LIN {X 0,Y 58.147,Z 234.055,A -85,B 0,C 180,E1 -29041.086,E2 -29041.086} C_VEL
LIN {X 0,Y 58.532,Z 233.998,A -85,B 0,C 180,E1 -29053.833,E2 -29053.833} C_VEL
LIN {X 0,Y 58.812,Z 233.964,A -85,B 0,C 180,E1 -29063.136,E2 -29063.136} C_VEL
LIN {X 0,Y 59.332,Z 233.898,A -85,B 0,C 180,E1 -29069.999,E2 -29069.999} C_VEL
LIN {X 0,Y 59.001,Z 234.006,A -85,B 0,C 180,E1 -29073.2,E2 -29073.2} C_VEL
LIN {X 0,Y 60.875,Z 241.106,A -85,B 0,C 180,E1 -29076.628,E2 -29076.628} C_VEL
LIN {X 0,Y 61.421,Z 249.605,A -85,B 0,C 180,E1 -29080.715,E2 -29080.715} C_VEL
LIN {X 0,Y 61.771,Z 259.733,A -85,B 0,C 180,E1 -29086.524,E2 -29086.524} C_VEL
LIN {X 0,Y 59.443,Z 268.589,A -85,B 0,C 180,E1 -29092.592,E2 -29092.592} C_VEL
LIN {X 0,Y 57.484,Z 276.014,A -85,B 0,C 180,E1 -29099.276,E2 -29099.276} C_VEL
LIN {X 0,Y 56.132,Z 282.39,A -85,B 0,C 180,E1 -29106.678,E2 -29106.678} C_VEL
LIN {X 0,Y 55.622,Z 288.326,A -85,B 0,C 180,E1 -29115.356,E2 -29115.356} C_VEL
LIN {X 0,Y 56.401,Z 293.902,A -85,B 0,C 180,E1 -29125.519,E2 -29125.519} C_VEL
LIN {X 0,Y 58.844,Z 298.13,A -85,B 0,C 180,E1 -29135.112,E2 -29135.112} C_VEL
LIN {X 0,Y 62.731,Z 301.206,A -85,B 0,C 180,E1 -29143.717,E2 -29143.717} C_VEL
LIN {X 0,Y 65.186,Z 302.377,A -85,B 0,C 180,E1 -29147.553,E2 -29147.553} C_VEL
LIN {X 0,Y 69.185,Z 303.56,A -85,B 0,C 180,E1 -29152.557,E2 -29152.557} C_VEL
LIN {X 0,Y 71.068,Z 304.167,A -85,B 0,C 180,E1 -29155.394,E2 -29155.394} C_VEL
LIN {X 0,Y 73.084,Z 304.818,A -85,B 0,C 180,E1 -29160.5,E2 -29160.5} C_VEL
LIN {X 0,Y 75.674,Z 305.088,A -85,B 0,C 180,E1 -29165.303,E2 -29165.303} C_VEL
LIN {X 0,Y 78.302,Z 305.043,A -85,B 0,C 180,E1 -29167.536,E2 -29167.536} C_VEL
LIN {X 0,Y 86.056,Z 304.44,A -85,B 0,C 180,E1 -29171.478,E2 -29171.478} C_VEL
LIN {X 0,Y 87.267,Z 304.356,A -85,B 0,C 180,E1 -29173.985,E2 -29173.985} C_VEL
LIN {X 0,Y 87.254,Z 304.599,A -85,B 0,C 180,E1 -29178.799,E2 -29178.799} C_VEL
LIN {X 0,Y 86.938,Z 305.009,A -85,B 0,C 180,E1 -29183.845,E2 -29183.845} C_VEL
LIN {X 0,Y 86.523,Z 305.313,A -85,B 0,C 180,E1 -29186.685,E2 -29186.685} C_VEL
LIN {X 0,Y 85.779,Z 305.678,A -85,B 0,C 180,E1 -29189.449,E2 -29189.449} C_VEL
LIN {X 0,Y 82.562,Z 306.32,A -85,B 0,C 180,E1 -29191.655,E2 -29191.655} C_VEL
LIN {X 0,Y 76.874,Z 306.876,A -85,B 0,C 180,E1 -29194.635,E2 -29194.635} C_VEL
LIN {X 0,Y 66.462,Z 306.835,A -85,B 0,C 180,E1 -29202.252,E2 -29202.252} C_VEL
LIN {X 0,Y 61.77,Z 306.092,A -85,B 0,C 180,E1 -29206.949,E2 -29206.949} C_VEL
LIN {X 0,Y 57.805,Z 304.93,A -85,B 0,C 180,E1 -29212.563,E2 -29212.563} C_VEL
LIN {X 0,Y 53.214,Z 302.399,A -85,B 0,C 180,E1 -29222.469,E2 -29222.469} C_VEL
LIN {X 0,Y 50.575,Z 298.791,A -85,B 0,C 180,E1 -29233.865,E2 -29233.865} C_VEL
LIN {X 0,Y 50.036,Z 293.872,A -85,B 0,C 180,E1 -29245.974,E2 -29245.974} C_VEL
LIN {X 0,Y 49.816,Z 288.545,A -85,B 0,C 180,E1 -29255.483,E2 -29255.483} C_VEL
LIN {X 0,Y 50.428,Z 282.817,A -85,B 0,C 180,E1 -29263.704,E2 -29263.704} C_VEL
LIN {X 0,Y 51.962,Z 275.543,A -85,B 0,C 180,E1 -29271.837,E2 -29271.837} C_VEL
LIN {X 0,Y 52.516,Z 271.35,A -85,B 0,C 180,E1 -29275.783,E2 -29275.783} C_VEL
LIN {X 0,Y 53.107,Z 261.909,A -85,B 0,C 180,E1 -29282.979,E2 -29282.979} C_VEL
LIN {X 0,Y 53.75,Z 253.089,A -85,B 0,C 180,E1 -29288.314,E2 -29288.314} C_VEL
LIN {X 0,Y 54.341,Z 243.271,A -85,B 0,C 180,E1 -29292.972,E2 -29292.972} C_VEL
LIN {X 0,Y 54.24,Z 241.536,A -85,B 0,C 180,E1 -29293.788,E2 -29293.788} C_VEL
LIN {X 0,Y 51.257,Z 235.226,A -85,B 0,C 180,E1 -29297.691,E2 -29297.691} C_VEL
LIN {X 0,Y 51.188,Z 234.914,A -85,B 0,C 180,E1 -29297.945,E2 -29297.945} C_VEL
LIN {X 0,Y 51.071,Z 234.929,A -85,B 0,C 180,E1 -29306.594,E2 -29306.594} C_VEL
LIN {X 0,Y 51.027,Z 234.937,A -85,B 0,C 180,E1 -29315.588,E2 -29315.588} C_VEL
LIN {X 0,Y 51.461,Z 234.884,A -85,B 0,C 180,E1 -29324.142,E2 -29324.142} C_VEL
LIN {X 0,Y 51.68,Z 234.856,A -85,B 0,C 180,E1 -29332.177,E2 -29332.177} C_VEL
LIN {X 0,Y 52.265,Z 234.781,A -85,B 0,C 180,E1 -29339.993,E2 -29339.993} C_VEL
LIN {X 0,Y 51.66,Z 234.855,A -85,B 0,C 180,E1 -29347.812,E2 -29347.812} C_VEL
LIN {X 0,Y 51.336,Z 234.896,A -85,B 0,C 180,E1 -29356.594,E2 -29356.594} C_VEL
LIN {X 0,Y 51.015,Z 234.935,A -85,B 0,C 180,E1 -29364.404,E2 -29364.404} C_VEL
LIN {X 0,Y 51.03,Z 234.938,A -85,B 0,C 180,E1 -29374.273,E2 -29374.273} C_VEL
LIN {X 0,Y 50.982,Z 234.942,A -85,B 0,C 180,E1 -29386.426,E2 -29386.426} C_VEL
LIN {X 0,Y 51.046,Z 234.93,A -85,B 0,C 180,E1 -29396.582,E2 -29396.582} C_VEL
LIN {X 0,Y 51.021,Z 234.933,A -85,B 0,C 180,E1 -29405.59,E2 -29405.59} C_VEL
LIN {X 0,Y 51.476,Z 234.877,A -85,B 0,C 180,E1 -29414.152,E2 -29414.152} C_VEL
LIN {X 0,Y 51.69,Z 234.85,A -85,B 0,C 180,E1 -29422.184,E2 -29422.184} C_VEL
LIN {X 0,Y 52.229,Z 234.783,A -85,B 0,C 180,E1 -29429.999,E2 -29429.999} C_VEL
LIN {X 0,Y 54.236,Z 242.713,A -85,B 0,C 180,E1 -29434.644,E2 -29434.644} C_VEL
LIN {X 0,Y 54.678,Z 252.656,A -85,B 0,C 180,E1 -29440.178,E2 -29440.178} C_VEL
LIN {X 0,Y 54.809,Z 259.647,A -85,B 0,C 180,E1 -29444.858,E2 -29444.858} C_VEL
LIN {X 0,Y 52.239,Z 269.02,A -85,B 0,C 180,E1 -29452.097,E2 -29452.097} C_VEL
LIN {X 0,Y 50.302,Z 276.011,A -85,B 0,C 180,E1 -29459.274,E2 -29459.274} C_VEL
LIN {X 0,Y 48.973,Z 282.317,A -85,B 0,C 180,E1 -29467.581,E2 -29467.581} C_VEL
LIN {X 0,Y 48.657,Z 288.871,A -85,B 0,C 180,E1 -29478.547,E2 -29478.547} C_VEL
LIN {X 0,Y 50.519,Z 295.238,A -85,B 0,C 180,E1 -29492.044,E2 -29492.044} C_VEL
LIN {X 0,Y 54.084,Z 299.168,A -85,B 0,C 180,E1 -29502.25,E2 -29502.25} C_VEL
LIN {X 0,Y 57.39,Z 301.314,A -85,B 0,C 180,E1 -29508.427,E2 -29508.427} C_VEL
LIN {X 0,Y 63.671,Z 303.578,A -85,B 0,C 180,E1 -29516.397,E2 -29516.397} C_VEL
LIN {X 0,Y 70.337,Z 304.754,A -85,B 0,C 180,E1 -29522.327,E2 -29522.327} C_VEL
LIN {X 0,Y 78.302,Z 305.043,A -85,B 0,C 180,E1 -29527.536,E2 -29527.536} C_VEL
LIN {X 0,Y 79.803,Z 305.04,A -85,B 0,C 180,E1 -29529.132,E2 -29529.132} C_VEL
LIN {X 0,Y 80.355,Z 305.113,A -85,B 0,C 180,E1 -29531.072,E2 -29531.072} C_VEL
LIN {X 0,Y 80.232,Z 305.361,A -85,B 0,C 180,E1 -29535.365,E2 -29535.365} C_VEL
LIN {X 0,Y 80.04,Z 305.687,A -85,B 0,C 180,E1 -29540.567,E2 -29540.567} C_VEL
LIN {X 0,Y 79.46,Z 306.136,A -85,B 0,C 180,E1 -29546.251,E2 -29546.251} C_VEL
LIN {X 0,Y 78.971,Z 306.223,A -85,B 0,C 180,E1 -29547.135,E2 -29547.135} C_VEL
LIN {X 0,Y 73.073,Z 306.664,A -85,B 0,C 180,E1 -29550.051,E2 -29550.051} C_VEL
LIN {X 0,Y 61.928,Z 306.166,A -85,B 0,C 180,E1 -29557.402,E2 -29557.402} C_VEL
LIN {X 0,Y 56.81,Z 305.332,A -85,B 0,C 180,E1 -29562.077,E2 -29562.077} C_VEL
LIN {X 0,Y 52.37,Z 304.024,A -85,B 0,C 180,E1 -29567.858,E2 -29567.858} C_VEL
LIN {X 0,Y 47.099,Z 301.265,A -85,B 0,C 180,E1 -29578.517,E2 -29578.517} C_VEL
LIN {X 0,Y 43.936,Z 297.328,A -85,B 0,C 180,E1 -29591.344,E2 -29591.344} C_VEL
LIN {X 0,Y 43.202,Z 293.068,A -85,B 0,C 180,E1 -29602.994,E2 -29602.994} C_VEL
LIN {X 0,Y 42.952,Z 289.875,A -85,B 0,C 180,E1 -29610.002,E2 -29610.002} C_VEL
LIN {X 0,Y 43.194,Z 283.298,A -85,B 0,C 180,E1 -29621.56,E2 -29621.56} C_VEL
LIN {X 0,Y 44.503,Z 276.476,A -85,B 0,C 180,E1 -29630.815,E2 -29630.815} C_VEL
LIN {X 0,Y 45.372,Z 272.557,A -85,B 0,C 180,E1 -29635.214,E2 -29635.214} C_VEL
LIN {X 0,Y 46.014,Z 263.487,A -85,B 0,C 180,E1 -29643.621,E2 -29643.621} C_VEL
LIN {X 0,Y 46.923,Z 254.054,A -85,B 0,C 180,E1 -29650.33,E2 -29650.33} C_VEL
LIN {X 0,Y 47.754,Z 244.411,A -85,B 0,C 180,E1 -29655.639,E2 -29655.639} C_VEL
LIN {X 0,Y 44.892,Z 238.404,A -85,B 0,C 180,E1 -29660.496,E2 -29660.496} C_VEL
LIN {X 0,Y 44.009,Z 235.811,A -85,B 0,C 180,E1 -29662.514,E2 -29662.514} C_VEL
LIN {X 0,Y 43.855,Z 235.829,A -85,B 0,C 180,E1 -29671.256,E2 -29671.256} C_VEL
LIN {X 0,Y 44.232,Z 235.779,A -85,B 0,C 180,E1 -29682.434,E2 -29682.434} C_VEL
LIN {X 0,Y 44.533,Z 235.742,A -85,B 0,C 180,E1 -29690.912,E2 -29690.912} C_VEL
LIN {X 0,Y 45.137,Z 235.668,A -85,B 0,C 180,E1 -29699.992,E2 -29699.992} C_VEL
LIN {X 0,Y 44.507,Z 235.749,A -85,B 0,C 180,E1 -29709.078,E2 -29709.078} C_VEL
LIN {X 0,Y 44.128,Z 235.801,A -85,B 0,C 180,E1 -29718.566,E2 -29718.566} C_VEL
LIN {X 0,Y 43.839,Z 235.834,A -85,B 0,C 180,E1 -29728.738,E2 -29728.738} C_VEL
LIN {X 0,Y 43.803,Z 235.832,A -85,B 0,C 180,E1 -29739.914,E2 -29739.914} C_VEL
LIN {X 0,Y 43.839,Z 235.836,A -85,B 0,C 180,E1 -29753.267,E2 -29753.267} C_VEL
LIN {X 0,Y 43.839,Z 235.837,A -85,B 0,C 180,E1 -29761.251,E2 -29761.251} C_VEL
LIN {X 0,Y 44.252,Z 235.777,A -85,B 0,C 180,E1 -29772.317,E2 -29772.317} C_VEL
LIN {X 0,Y 44.736,Z 235.723,A -85,B 0,C 180,E1 -29784.929,E2 -29784.929} C_VEL
LIN {X 0,Y 44.742,Z 235.725,A -85,B 0,C 180,E1 -29785.494,E2 -29785.494} C_VEL
LIN {X 0,Y 45.948,Z 238.577,A -85,B 0,C 180,E1 -29787.807,E2 -29787.807} C_VEL
LIN {X 0,Y 46.921,Z 241.271,A -85,B 0,C 180,E1 -29789.998,E2 -29789.998} C_VEL
LIN {X 0,Y 47.82,Z 245.986,A -85,B 0,C 180,E1 -29793.158,E2 -29793.158} C_VEL
LIN {X 0,Y 47.853,Z 255.286,A -85,B 0,C 180,E1 -29799.509,E2 -29799.509} C_VEL
LIN {X 0,Y 47.627,Z 260.954,A -85,B 0,C 180,E1 -29803.873,E2 -29803.873} C_VEL
LIN {X 0,Y 44.732,Z 270.214,A -85,B 0,C 180,E1 -29812.319,E2 -29812.319} C_VEL
LIN {X 0,Y 42.707,Z 277.644,A -85,B 0,C 180,E1 -29821.567,E2 -29821.567} C_VEL
LIN {X 0,Y 41.638,Z 284.323,A -85,B 0,C 180,E1 -29832.464,E2 -29832.464} C_VEL
LIN {X 0,Y 42.252,Z 290.948,A -85,B 0,C 180,E1 -29846.268,E2 -29846.268} C_VEL
LIN {X 0,Y 45.126,Z 296.053,A -85,B 0,C 180,E1 -29859.136,E2 -29859.136} C_VEL
LIN {X 0,Y 49.944,Z 299.969,A -85,B 0,C 180,E1 -29870.066,E2 -29870.066} C_VEL
LIN {X 0,Y 57.56,Z 303.224,A -85,B 0,C 180,E1 -29880.006,E2 -29880.006} C_VEL
LIN {X 0,Y 64.843,Z 304.812,A -85,B 0,C 180,E1 -29886.227,E2 -29886.227} C_VEL
LIN {X 0,Y 74.163,Z 305.46,A -85,B 0,C 180,E1 -29891.858,E2 -29891.858} C_VEL
LIN {X 0,Y 79.864,Z 305.337,A -85,B 0,C 180,E1 -29894.539,E2 -29894.539} C_VEL
LIN {X 0,Y 80.232,Z 305.361,A -85,B 0,C 180,E1 -29895.365,E2 -29895.365} C_VEL
LIN {X 0,Y 79.457,Z 305.55,A -85,B 0,C 180,E1 -29897.626,E2 -29897.626} C_VEL
LIN {X 0,Y 77.306,Z 305.831,A -85,B 0,C 180,E1 -29900.075,E2 -29900.075} C_VEL
LIN {X 0,Y 73.783,Z 306.13,A -85,B 0,C 180,E1 -29902.59,E2 -29902.59} C_VEL
LIN {X 0,Y 70.196,Z 306.297,A -85,B 0,C 180,E1 -29904.632,E2 -29904.632} C_VEL
LIN {X 0,Y 65.203,Z 306.186,A -85,B 0,C 180,E1 -29907.293,E2 -29907.293} C_VEL
LIN {X 0,Y 57.906,Z 305.483,A -85,B 0,C 180,E1 -29911.836,E2 -29911.836} C_VEL
LIN {X 0,Y 52.348,Z 304.427,A -85,B 0,C 180,E1 -29916.341,E2 -29916.341} C_VEL
LIN {X 0,Y 47.389,Z 302.996,A -85,B 0,C 180,E1 -29922.141,E2 -29922.141} C_VEL
LIN {X 0,Y 41.31,Z 299.905,A -85,B 0,C 180,E1 -29933.458,E2 -29933.458} C_VEL
LIN {X 0,Y 37.452,Z 295.707,A -85,B 0,C 180,E1 -29947.959,E2 -29947.959} C_VEL
LIN {X 0,Y 36.406,Z 291.241,A -85,B 0,C 180,E1 -29961.677,E2 -29961.677} C_VEL
LIN {X 0,Y 35.976,Z 287.808,A -85,B 0,C 180,E1 -29970.002,E2 -29970.002} C_VEL
LIN {X 0,Y 36.18,Z 282.253,A -85,B 0,C 180,E1 -29981.203,E2 -29981.203} C_VEL
LIN {X 0,Y 37.549,Z 275.454,A -85,B 0,C 180,E1 -29991.985,E2 -29991.985} C_VEL
LIN {X 0,Y 38.405,Z 271.463,A -85,B 0,C 180,E1 -29997.227,E2 -29997.227} C_VEL
LIN {X 0,Y 39.317,Z 262.055,A -85,B 0,C 180,E1 -30007.108,E2 -30007.108} C_VEL
LIN {X 0,Y 40.363,Z 253.404,A -85,B 0,C 180,E1 -30014.148,E2 -30014.148} C_VEL
LIN {X 0,Y 41.159,Z 246.849,A -85,B 0,C 180,E1 -30018.428,E2 -30018.428} C_VEL
LIN {X 0,Y 38.746,Z 241.031,A -85,B 0,C 180,E1 -30024.38,E2 -30024.38} C_VEL
LIN {X 0,Y 36.902,Z 237.45,A -85,B 0,C 180,E1 -30028.406,E2 -30028.406} C_VEL
LIN {X 0,Y 36.786,Z 236.716,A -85,B 0,C 180,E1 -30029.096,E2 -30029.096} C_VEL
LIN {X 0,Y 37.059,Z 236.672,A -85,B 0,C 180,E1 -30041.487,E2 -30041.487} C_VEL
LIN {X 0,Y 37.33,Z 236.638,A -85,B 0,C 180,E1 -30049.139,E2 -30049.139} C_VEL
LIN {X 0,Y 37.992,Z 236.557,A -85,B 0,C 180,E1 -30059.991,E2 -30059.991} C_VEL
LIN {X 0,Y 37.302,Z 236.651,A -85,B 0,C 180,E1 -30070.85,E2 -30070.85} C_VEL
LIN {X 0,Y 37.041,Z 236.682,A -85,B 0,C 180,E1 -30078.429,E2 -30078.429} C_VEL
LIN {X 0,Y 36.721,Z 236.721,A -85,B 0,C 180,E1 -30095.03,E2 -30095.03} C_VEL
LIN {X 0,Y 36.723,Z 236.713,A -85,B 0,C 180,E1 -30100.044,E2 -30100.044} C_VEL
LIN {X 0,Y 36.721,Z 236.715,A -85,B 0,C 180,E1 -30109.94,E2 -30109.94} C_VEL
LIN {X 0,Y 36.718,Z 236.716,A -85,B 0,C 180,E1 -30114.952,E2 -30114.952} C_VEL
LIN {X 0,Y 37.075,Z 236.673,A -85,B 0,C 180,E1 -30131.378,E2 -30131.378} C_VEL
LIN {X 0,Y 37.354,Z 236.746,A -85,B 0,C 180,E1 -30139.153,E2 -30139.153} C_VEL
LIN {X 0,Y 38.514,Z 239.392,A -85,B 0,C 180,E1 -30142.132,E2 -30142.132} C_VEL
LIN {X 0,Y 40.4,Z 242.862,A -85,B 0,C 180,E1 -30146.258,E2 -30146.258} C_VEL
LIN {X 0,Y 41.268,Z 247.314,A -85,B 0,C 180,E1 -30149.998,E2 -30149.998} C_VEL
LIN {X 0,Y 41.051,Z 256.473,A -85,B 0,C 180,E1 -30157.375,E2 -30157.375} C_VEL
LIN {X 0,Y 40.845,Z 260.704,A -85,B 0,C 180,E1 -30161.16,E2 -30161.16} C_VEL
LIN {X 0,Y 37.64,Z 270.122,A -85,B 0,C 180,E1 -30171.028,E2 -30171.028} C_VEL
LIN {X 0,Y 35.651,Z 276.967,A -85,B 0,C 180,E1 -30181.04,E2 -30181.04} C_VEL
LIN {X 0,Y 34.697,Z 282.312,A -85,B 0,C 180,E1 -30191.054,E2 -30191.054} C_VEL
LIN {X 0,Y 34.909,Z 287.813,A -85,B 0,C 180,E1 -30203.635,E2 -30203.635} C_VEL
LIN {X 0,Y 37.157,Z 293.187,A -85,B 0,C 180,E1 -30217.783,E2 -30217.783} C_VEL
LIN {X 0,Y 41.617,Z 297.687,A -85,B 0,C 180,E1 -30230.286,E2 -30230.286} C_VEL
LIN {X 0,Y 49.219,Z 301.788,A -85,B 0,C 180,E1 -30241.814,E2 -30241.814} C_VEL
LIN {X 0,Y 56.902,Z 304.094,A -85,B 0,C 180,E1 -30248.864,E2 -30248.864} C_VEL
LIN {X 0,Y 65.212,Z 305.427,A -85,B 0,C 180,E1 -30254.088,E2 -30254.088} C_VEL
LIN {X 0,Y 71.596,Z 305.87,A -85,B 0,C 180,E1 -30257.131,E2 -30257.131} C_VEL
LIN {X 0,Y 72.946,Z 305.989,A -85,B 0,C 180,E1 -30259.712,E2 -30259.712} C_VEL
LIN {X 0,Y 72.629,Z 306.194,A -85,B 0,C 180,E1 -30262.777,E2 -30262.777} C_VEL
LIN {X 0,Y 69.785,Z 306.297,A -85,B 0,C 180,E1 -30264.992,E2 -30264.992} C_VEL
LIN {X 0,Y 65.203,Z 306.186,A -85,B 0,C 180,E1 -30267.293,E2 -30267.293} C_VEL
LIN {X 0,Y 59.927,Z 305.785,A -85,B 0,C 180,E1 -30269.696,E2 -30269.696} C_VEL
LIN {X 0,Y 50.679,Z 304.107,A -85,B 0,C 180,E1 -30273.001,E2 -30273.001} C_VEL
LIN {X 0,Y 41.943,Z 301.476,A -85,B 0,C 180,E1 -30277.797,E2 -30277.797} C_VEL
LIN {X 0,Y 37.745,Z 299.578,A -85,B 0,C 180,E1 -30283.092,E2 -30283.092} C_VEL
LIN {X 0,Y 32.448,Z 295.659,A -85,B 0,C 180,E1 -30297.218,E2 -30297.218} C_VEL
LIN {X 0,Y 30.047,Z 291.371,A -85,B 0,C 180,E1 -30312.772,E2 -30312.772} C_VEL
LIN {X 0,Y 29.428,Z 288.175,A -85,B 0,C 180,E1 -30323.145,E2 -30323.145} C_VEL
LIN {X 0,Y 29.164,Z 281.322,A -85,B 0,C 180,E1 -30340.276,E2 -30340.276} C_VEL
LIN {X 0,Y 30.591,Z 274.515,A -85,B 0,C 180,E1 -30353.479,E2 -30353.479} C_VEL
LIN {X 0,Y 31.345,Z 271.428,A -85,B 0,C 180,E1 -30358.457,E2 -30358.457} C_VEL
LIN {X 0,Y 32.52,Z 262.097,A -85,B 0,C 180,E1 -30370.42,E2 -30370.42} C_VEL
LIN {X 0,Y 34.001,Z 252.847,A -85,B 0,C 180,E1 -30379.257,E2 -30379.257} C_VEL
LIN {X 0,Y 34.693,Z 248.698,A -85,B 0,C 180,E1 -30382.562,E2 -30382.562} C_VEL
LIN {X 0,Y 31.313,Z 241.237,A -85,B 0,C 180,E1 -30393.316,E2 -30393.316} C_VEL
LIN {X 0,Y 29.959,Z 238.453,A -85,B 0,C 180,E1 -30398.179,E2 -30398.179} C_VEL
LIN {X 0,Y 29.838,Z 237.453,A -85,B 0,C 180,E1 -30399.383,E2 -30399.383} C_VEL
LIN {X 0,Y 30.108,Z 237.429,A -85,B 0,C 180,E1 -30406.49,E2 -30406.49} C_VEL
LIN {X 0,Y 30.806,Z 237.361,A -85,B 0,C 180,E1 -30419.989,E2 -30419.989} C_VEL
LIN {X 0,Y 30.086,Z 237.429,A -85,B 0,C 180,E1 -30433.497,E2 -30433.497} C_VEL
LIN {X 0,Y 29.852,Z 237.453,A -85,B 0,C 180,E1 -30439.65,E2 -30439.65} C_VEL
LIN {X 0,Y 29.489,Z 237.486,A -85,B 0,C 180,E1 -30448.453,E2 -30448.453} C_VEL
LIN {X 0,Y 29.538,Z 237.482,A -85,B 0,C 180,E1 -30465.527,E2 -30465.527} C_VEL
LIN {X 0,Y 29.504,Z 237.485,A -85,B 0,C 180,E1 -30481.545,E2 -30481.545} C_VEL
LIN {X 0,Y 29.751,Z 237.462,A -85,B 0,C 180,E1 -30487.813,E2 -30487.813} C_VEL
LIN {X 0,Y 30.612,Z 239.685,A -85,B 0,C 180,E1 -30491.68,E2 -30491.68} C_VEL
LIN {X 0,Y 33.078,Z 243.608,A -85,B 0,C 180,E1 -30499.283,E2 -30499.283} C_VEL
LIN {X 0,Y 34.266,Z 245.862,A -85,B 0,C 180,E1 -30502.633,E2 -30502.633} C_VEL
LIN {X 0,Y 34.79,Z 248.449,A -85,B 0,C 180,E1 -30505.653,E2 -30505.653} C_VEL
LIN {X 0,Y 34.406,Z 256.029,A -85,B 0,C 180,E1 -30512.925,E2 -30512.925} C_VEL
LIN {X 0,Y 34.138,Z 260.204,A -85,B 0,C 180,E1 -30517.39,E2 -30517.39} C_VEL
LIN {X 0,Y 30.598,Z 269.837,A -85,B 0,C 180,E1 -30529.061,E2 -30529.061} C_VEL
LIN {X 0,Y 28.538,Z 276.459,A -85,B 0,C 180,E1 -30540.75,E2 -30540.75} C_VEL
LIN {X 0,Y 27.63,Z 282.856,A -85,B 0,C 180,E1 -30555.821,E2 -30555.821} C_VEL
LIN {X 0,Y 28.5,Z 288.043,A -85,B 0,C 180,E1 -30570.463,E2 -30570.463} C_VEL
LIN {X 0,Y 31.029,Z 292.416,A -85,B 0,C 180,E1 -30583.613,E2 -30583.613} C_VEL
LIN {X 0,Y 35.268,Z 296.342,A -85,B 0,C 180,E1 -30595.096,E2 -30595.096} C_VEL
LIN {X 0,Y 42.4,Z 300.329,A -85,B 0,C 180,E1 -30606.016,E2 -30606.016} C_VEL
LIN {X 0,Y 53.362,Z 303.989,A -85,B 0,C 180,E1 -30615.279,E2 -30615.279} C_VEL
LIN {X 0,Y 62.117,Z 305.573,A -85,B 0,C 180,E1 -30619.848,E2 -30619.848} C_VEL
LIN {X 0,Y 60.729,Z 305.516,A -85,B 0,C 180,E1 -30622.21,E2 -30622.21} C_VEL
LIN {X 0,Y 54.509,Z 304.772,A -85,B 0,C 180,E1 -30625.51,E2 -30625.51} C_VEL
LIN {X 0,Y 48.507,Z 303.487,A -85,B 0,C 180,E1 -30629.623,E2 -30629.623} C_VEL
LIN {X 0,Y 38.091,Z 299.774,A -85,B 0,C 180,E1 -30642.44,E2 -30642.44} C_VEL
LIN {X 0,Y 37.745,Z 299.578,A -85,B 0,C 180,E1 -30643.092,E2 -30643.092} C_VEL
LIN {X 0,Y 34.146,Z 297.51,A -85,B 0,C 180,E1 -30649.648,E2 -30649.648} C_VEL
LIN {X 0,Y 30.463,Z 294.926,A -85,B 0,C 180,E1 -30656.467,E2 -30656.467} C_VEL
LIN {X 0,Y 24.122,Z 288.564,A -85,B 0,C 180,E1 -30673.455,E2 -30673.455} C_VEL
LIN {X 0,Y 22.151,Z 283.599,A -85,B 0,C 180,E1 -30688.882,E2 -30688.882} C_VEL
LIN {X 0,Y 22.958,Z 275.965,A -85,B 0,C 180,E1 -30710.333,E2 -30710.333} C_VEL
LIN {X 0,Y 24.357,Z 270.922,A -85,B 0,C 180,E1 -30720.98,E2 -30720.98} C_VEL
LIN {X 0,Y 25.891,Z 261.93,A -85,B 0,C 180,E1 -30735.446,E2 -30735.446} C_VEL
LIN {X 0,Y 27.959,Z 252.372,A -85,B 0,C 180,E1 -30746.338,E2 -30746.338} C_VEL
LIN {X 0,Y 28.227,Z 250.811,A -85,B 0,C 180,E1 -30747.924,E2 -30747.924} C_VEL
LIN {X 0,Y 25.916,Z 244.959,A -85,B 0,C 180,E1 -30759.669,E2 -30759.669} C_VEL
LIN {X 0,Y 24.658,Z 241.953,A -85,B 0,C 180,E1 -30767.643,E2 -30767.643} C_VEL
LIN {X 0,Y 23.6,Z 239.648,A -85,B 0,C 180,E1 -30775.716,E2 -30775.716} C_VEL
LIN {X 0,Y 23.575,Z 237.854,A -85,B 0,C 180,E1 -30779.985,E2 -30779.985} C_VEL
LIN {X 0,Y 22.796,Z 237.878,A -85,B 0,C 180,E1 -30797.941,E2 -30797.941} C_VEL
LIN {X 0,Y 22.162,Z 237.897,A -85,B 0,C 180,E1 -30817.682,E2 -30817.682} C_VEL
LIN {X 0,Y 25.585,Z 243.842,A -85,B 0,C 180,E1 -30845.897,E2 -30845.897} C_VEL
LIN {X 0,Y 28.406,Z 249.235,A -85,B 0,C 180,E1 -30858.626,E2 -30858.626} C_VEL
LIN {X 0,Y 28.534,Z 251.417,A -85,B 0,C 180,E1 -30861.582,E2 -30861.582} C_VEL
LIN {X 0,Y 27.541,Z 259.741,A -85,B 0,C 180,E1 -30871.825,E2 -30871.825} C_VEL
LIN {X 0,Y 25.722,Z 264.466,A -85,B 0,C 180,E1 -30877.849,E2 -30877.849} C_VEL
LIN {X 0,Y 22.61,Z 272.118,A -85,B 0,C 180,E1 -30891.217,E2 -30891.217} C_VEL
LIN {X 0,Y 20.818,Z 278.765,A -85,B 0,C 180,E1 -30908.614,E2 -30908.614} C_VEL
LIN {X 0,Y 21.29,Z 285.062,A -85,B 0,C 180,E1 -30929.911,E2 -30929.911} C_VEL
LIN {X 0,Y 25.324,Z 291.491,A -85,B 0,C 180,E1 -30952.046,E2 -30952.046} C_VEL
LIN {X 0,Y 31.782,Z 296.422,A -85,B 0,C 180,E1 -30966.359,E2 -30966.359} C_VEL
LIN {X 0,Y 39.853,Z 300.365,A -85,B 0,C 180,E1 -30975.578,E2 -30975.578} C_VEL
LIN {X 0,Y 44.644,Z 302.128,A -85,B 0,C 180,E1 -30979.175,E2 -30979.175} C_VEL
LIN {X 0,Y 45.442,Z 302.503,A -85,B 0,C 180,E1 -30981.885,E2 -30981.885} C_VEL
LIN {X 0,Y 36.51,Z 299.562,A -85,B 0,C 180,E1 -30989.981,E2 -30989.981} C_VEL
LIN {X 0,Y 28.929,Z 295.56,A -85,B 0,C 180,E1 -31003.216,E2 -31003.216} C_VEL
LIN {X 0,Y 24.951,Z 291.905,A -85,B 0,C 180,E1 -31017.7,E2 -31017.7} C_VEL
LIN {X 0,Y 22.944,Z 287.19,A -85,B 0,C 180,E1 -31036.722,E2 -31036.722} C_VEL
LIN {X 0,Y 22.151,Z 283.599,A -85,B 0,C 180,E1 -31048.882,E2 -31048.882} C_VEL
LIN {X 0,Y 21.76,Z 281.082,A -85,B 0,C 180,E1 -31056.724,E2 -31056.724} C_VEL
LIN {X 0,Y 20.806,Z 276.94,A -85,B 0,C 180,E1 -31067.912,E2 -31067.912} C_VEL
LIN {X 0,Y 19.793,Z 272.544,A -85,B 0,C 180,E1 -31079.05,E2 -31079.05} C_VEL
LIN {X 0,Y 19.423,Z 263.036,A -85,B 0,C 180,E1 -31101.397,E2 -31101.397} C_VEL
LIN {X 0,Y 20.232,Z 259.516,A -85,B 0,C 180,E1 -31107.39,E2 -31107.39} C_VEL
LIN {X 0,Y 22.096,Z 252.974,A -85,B 0,C 180,E1 -31116.272,E2 -31116.272} C_VEL
LIN {X 0,Y 20.864,Z 248.126,A -85,B 0,C 180,E1 -31130.287,E2 -31130.287} C_VEL
LIN {X 0,Y 20.065,Z 245.877,A -85,B 0,C 180,E1 -31139.983,E2 -31139.983} C_VEL
LIN {X 0,Y 19.609,Z 244.174,A -85,B 0,C 180,E1 -31150.306,E2 -31150.306} C_VEL
LIN {X 0,Y 19.288,Z 244.359,A -85,B 0,C 180,E1 -31173.123,E2 -31173.123} C_VEL
LIN {X 0,Y 20.99,Z 248.972,A -85,B 0,C 180,E1 -31200.685,E2 -31200.685} C_VEL
LIN {X 0,Y 22.434,Z 252.258,A -85,B 0,C 180,E1 -31211.74,E2 -31211.74} C_VEL
LIN {X 0,Y 22.515,Z 253.531,A -85,B 0,C 180,E1 -31214.148,E2 -31214.148} C_VEL
LIN {X 0,Y 21.183,Z 260.016,A -85,B 0,C 180,E1 -31224.284,E2 -31224.284} C_VEL
LIN {X 0,Y 17.003,Z 268.57,A -85,B 0,C 180,E1 -31238.912,E2 -31238.912} C_VEL
LIN {X 0,Y 13.909,Z 277.001,A -85,B 0,C 180,E1 -31266.91,E2 -31266.91} C_VEL
LIN {X 0,Y 14.992,Z 283.939,A -85,B 0,C 180,E1 -31299.637,E2 -31299.637} C_VEL
LIN {X 0,Y 20.224,Z 290.15,A -85,B 0,C 180,E1 -31324.159,E2 -31324.159} C_VEL
LIN {X 0,Y 28.28,Z 295.612,A -85,B 0,C 180,E1 -31338.082,E2 -31338.082} C_VEL
LIN {X 0,Y 29.873,Z 296.5,A -85,B 0,C 180,E1 -31339.78,E2 -31339.78} C_VEL
LIN {X 0,Y 30.487,Z 296.869,A -85,B 0,C 180,E1 -31342.772,E2 -31342.772} C_VEL
LIN {X 0,Y 21.947,Z 292.021,A -85,B 0,C 180,E1 -31358.326,E2 -31358.326} C_VEL
LIN {X 0,Y 16.929,Z 286.146,A -85,B 0,C 180,E1 -31385.476,E2 -31385.476} C_VEL
LIN {X 0,Y 15.263,Z 280.699,A -85,B 0,C 180,E1 -31410.005,E2 -31410.005} C_VEL
LIN {X 0,Y 16.269,Z 273.88,A -85,B 0,C 180,E1 -31435.599,E2 -31435.599} C_VEL
LIN {X 0,Y 17.49,Z 270.039,A -85,B 0,C 180,E1 -31446.489,E2 -31446.489} C_VEL
LIN {X 0,Y 19.828,Z 260.852,A -85,B 0,C 180,E1 -31465.318,E2 -31465.318} C_VEL
LIN {X 0,Y 20.232,Z 259.516,A -85,B 0,C 180,E1 -31467.39,E2 -31467.39} C_VEL
LIN {X 0,Y 20.153,Z 257.935,A -85,B 0,C 180,E1 -31471.026,E2 -31471.026} C_VEL
LIN {X 0,Y 18.988,Z 256.459,A -85,B 0,C 180,E1 -31477.504,E2 -31477.504} C_VEL
LIN {X 0,Y 16.56,Z 254.147,A -85,B 0,C 180,E1 -31493.979,E2 -31493.979} C_VEL
LIN {X 0,Y 16.452,Z 253.428,A -85,B 0,C 180,E1 -31497.368,E2 -31497.368} C_VEL
LIN {X 0,Y 16.466,Z 252.777,A -85,B 0,C 180,E1 -31499.979,E2 -31499.979} C_VEL
LIN {X 0,Y 16.379,Z 250.833,A -85,B 0,C 180,E1 -31512.367,E2 -31512.367} C_VEL
LIN {X 0,Y 16.167,Z 250.64,A -85,B 0,C 180,E1 -31525.743,E2 -31525.743} C_VEL
LIN {X 0,Y 16.718,Z 254.673,A -85,B 0,C 180,E1 -31557.181,E2 -31557.181} C_VEL
LIN {X 0,Y 16.891,Z 255.374,A -85,B 0,C 180,E1 -31560.535,E2 -31560.535} C_VEL
LIN {X 0,Y 15.982,Z 258.503,A -85,B 0,C 180,E1 -31567.368,E2 -31567.368} C_VEL
LIN {X 0,Y 15.558,Z 259.842,A -85,B 0,C 180,E1 -31570.122,E2 -31570.122} C_VEL
LIN {X 0,Y 11.837,Z 266.033,A -85,B 0,C 180,E1 -31580.596,E2 -31580.596} C_VEL
LIN {X 0,Y 7.545,Z 273.633,A -85,B 0,C 180,E1 -31611.465,E2 -31611.465} C_VEL
LIN {X 0,Y 9.465,Z 282.567,A -85,B 0,C 180,E1 -31680.036,E2 -31680.036} C_VEL
LIN {X 0,Y 17.342,Z 289.259,A -85,B 0,C 180,E1 -31703.929,E2 -31703.929} C_VEL
LIN {X 0,Y 11.129,Z 283.799,A -85,B 0,C 180,E1 -31730.846,E2 -31730.846} C_VEL
LIN {X 0,Y 8.419,Z 276.29,A -85,B 0,C 180,E1 -31782.056,E2 -31782.056} C_VEL
LIN {X 0,Y 10.432,Z 270.638,A -85,B 0,C 180,E1 -31812.365,E2 -31812.365} C_VEL
LIN {X 0,Y 14.171,Z 261.133,A -85,B 0,C 180,E1 -31839.936,E2 -31839.936} C_VEL
LIN {X 0,Y 16.352,Z 256.246,A -85,B 0,C 180,E1 -31847.838,E2 -31847.838} C_VEL
LIN {X 0,Y 16.527,Z 254.724,A -85,B 0,C 180,E1 -31852.18,E2 -31852.18} C_VEL
LIN {X 0,Y 16.452,Z 253.428,A -85,B 0,C 180,E1 -31857.368,E2 -31857.368} C_VEL
LIN {X 0,Y 16.014,Z 253.033,A -85,B 0,C 180,E1 -31862.723,E2 -31862.723} C_VEL
LIN {X 0,Y 14.833,Z 253.977,A -85,B 0,C 180,E1 -31870.914,E2 -31870.914} C_VEL
LIN {X 0,Y 12.965,Z 256.667,A -85,B 0,C 180,E1 -31881.133,E2 -31881.133} C_VEL
LIN {X 0,Y 10.508,Z 260.704,A -85,B 0,C 180,E1 -31890.244,E2 -31890.244} C_VEL
LIN {X 0,Y 7.669,Z 265.212,A -85,B 0,C 180,E1 -31899.612,E2 -31899.612} C_VEL
LIN {X 0,Y 4.402,Z 269.509,A -85,B 0,C 180,E1 -31906.097,E2 -31906.097} C_VEL
LIN {X 0,Y 0.039,Z 274.264,A -85,B 0,C 180,E1 -32048.865,E2 -32048.865} C_VEL
LIN {X 0,Y 1.513,Z 274.936,A -85,B 0,C 180,E1 -32130.05,E2 -32130.05} C_VEL
LIN {X 0,Y 5.341,Z 269.1,A -85,B 0,C 180,E1 -32210.782,E2 -32210.782} C_VEL
LIN {X 0,Y 11.24,Z 259.973,A -85,B 0,C 180,E1 -32229.847,E2 -32229.847} C_VEL
LIN {X 0,Y 12.409,Z 257.954,A -85,B 0,C 180,E1 -32232.234,E2 -32232.234} C_VEL
LIN {X 0,Y 12.631,Z 257.366,A -85,B 0,C 180,E1 -32236.124,E2 -32236.124} C_VEL
LIN {X 0,Y 12.071,Z 258.95,A -85,B 0,C 180,E1 -32261.355,E2 -32261.355} C_VEL
LIN {X 0,Y 11.344,Z 260.418,A -85,B 0,C 180,E1 -32264.831,E2 -32264.831} C_VEL
LIN {X 0,Y 4.402,Z 269.509,A -85,B 0,C 180,E1 -32266.097,E2 -32266.097} C_VEL
LIN {X 0,Y 3.909,Z 270.825,A -85,B 0,C 180,E1 -32266.384,E2 -32266.384} C_VEL
LIN {X 0,Y 3.909,Z 600,A -85,B 0,C 180,E1 -32266.384,E2 -32266.384} C_VEL
LIN {X 0,Y 3.909,Z 600,A -85,B 0,C 180,E1 -32266.384,E2 -32266.384}

QRS_NEXT_CUT()

QRS_NEXT()
QRS_HOME()

END
